{attribute wpf [Container(Layout.Stack)]}
TYPE stTreeStruct :
STRUCT
	One:BOOL;
	Two:BOOL;
	Another:STRING;
	ThisOne:STRING;
	ANumberWouldBeCool:INT;
	Bools : stBools;
END_STRUCT
END_TYPE

(* stored: Version 1.1.0.1, ProductVersion 3.1.4024.5
   DUT stTreeStruct: Id {c4f063bc-7fb2-4160-8cc1-8cee5dd4e4a4} *)
